(* Logix 5000 project; controller FPosB_EVO3_SP12 vendor 1 type 14 code 154 rev 30.11; software revision 30.01 *)
// v6: Studio5k 30+
// Works with CPX-E FW 1.1.24

TASK MainTask (continuous, watchdog 500 ms) : MainProgram

MODULES
   Local : vendor 1 type 14 code 154 (PointIO 0, rev 30.11)
      FMCP_Multi_EVO3_SP12 : ETHERNET-MODULE (Ethernet 192.168.4.20, rev 1.1, Output RPI 10 ms)
      Discrete_IO : Embedded (PointIO 1, rev 30.11, Output RPI 20 ms)
END_MODULES

ADD_ON_INSTRUCTION FMCP_Multi_EVO3_CPX_E_SP12_CPX_E   (* revision 3.14 15, vendor Festo Inc *)
// Multikinematic AOI to control up to 4 axis per kinematic and up to 3 different kinematics
// Revision note:
// 3.14.15: Multikinematic with 4 axis per kinematic
// 3.14.15: Additional tag to try to recover from a minor fault
VAR_IN_OUT
   InputData : DINT[64]; {required}
   OutputData : DINT[64]; {required}
END_VAR
VAR_INPUT
   K_I_N_E_M_A_T_I_C_1 : BOOL; {visible}
   I_n_p_u_t_s_K_1 : BOOL; {visible}
   sModeSelectorK1 : SINT; {visible}
END_VAR
VAR_OUTPUT
   sModeSelectedK1 : SINT; {visible}
END_VAR
VAR_INPUT
   rXAxisMove_CNCOffsetK1 : DINT; {visible}
   rYAxisMove_CNCOffsetK1 : DINT; {visible}
   rZAxisMove_CNCOffsetK1 : DINT; {visible}
   rUAxisMoveK1 : DINT; {visible}
   rZAxisOffset_CNCNumberK1 : DINT; {visible}
   rSmoothRad_CNCPhiK1 : DINT; {visible}
   rNominalVel_CNCConstantVelK1 : DINT := 1000; {visible}
   rLowVelMoveK1 : DINT := 100; {visible}
   rMoveAccelerationK1 : DINT := 1000; {visible}
   rMoveDecelerationK1 : DINT := 1000; {visible}
   rZAxisUpMoveK1 : DINT; {visible}
   bMoveK1 : BOOL; {visible}
   bJogXPosK1 : BOOL; {visible}
   bJogXNegK1 : BOOL; {visible}
   bJogYPosK1 : BOOL; {visible}
   bJogYNegK1 : BOOL; {visible}
   bJogZPosK1 : BOOL; {visible}
   bJogZNegK1 : BOOL; {visible}
   bJogUPosK1 : BOOL; {visible}
   bJogUNegK1 : BOOL; {visible}
   bAckMK1 : BOOL; {visible}
   bAckAllMK1 : BOOL; {visible}
   bHaltK1 : BOOL; {visible}
   bAbortMotionTaskK1 : BOOL; {visible}
   bTryToClearFaultK1 : BOOL; {visible}
   uOverrideK1 : DINT; {visible}
   O_u_t_p_u_t_s_K_1 : BOOL; {visible}
END_VAR
VAR_OUTPUT
   rXAxisActualPositionK1 : DINT; {visible}
   rYAxisActualPositionK1 : DINT; {visible}
   rZAxisActualPositionK1 : DINT; {visible}
   rUAxisActualPositionK1 : DINT; {visible}
   bEnabledK1 : BOOL; {visible}
   bHomedK1 : BOOL; {visible}
   bHaltedK1 : BOOL; {visible}
   bMoveDnK1 : BOOL; {visible}
   bMovingK1 : BOOL; {visible}
   bBusyK1 : BOOL; {visible}
   bErrorK1 : BOOL; {visible}
   bSafetyStatusK1 : BOOL; {visible}
   bMotionTaskAbortedK1 : BOOL; {visible}
   bXAxisSWLimitNegK1 : BOOL; {visible}
   bXAxisSWLimitPosK1 : BOOL; {visible}
   bYAxisSWLimitNegK1 : BOOL; {visible}
   bYAxisSWLimitPosK1 : BOOL; {visible}
   bZAxisSWLimitNegK1 : BOOL; {visible}
   bZAxisSWLimitPosK1 : BOOL; {visible}
   bUAxisSWLimitNegK1 : BOOL; {visible}
   bUAxisSWLimitPosK1 : BOOL; {visible}
   bHSwitchPoint1K1 : BOOL; {visible}
   bHSwitchPoint2K1 : BOOL; {visible}
   bMActiveK1 : BOOL; {visible}
   dErrorCode1K1 : DINT; {visible}
   dErrorCode2K1 : DINT; {visible}
   rGCodeLineK1 : DINT; {visible}
   bAtPrePickK1 : BOOL; {visible}
   bAtPickK1 : BOOL; {visible}
   bAtPrePlaceK1 : BOOL; {visible}
   bAtPlaceK1 : BOOL; {visible}
END_VAR
VAR_INPUT
   K_I_N_E_M_A_T_I_C_2 : BOOL; {visible}
   I_n_p_u_t_s_K_2 : BOOL; {visible}
   sModeSelectorK2 : SINT; {visible}
END_VAR
VAR_OUTPUT
   sModeSelectedK2 : SINT; {visible}
END_VAR
VAR_INPUT
   rXAxisMove_CNCOffsetK2 : DINT;
   rYAxisMove_CNCOffsetK2 : DINT; {visible}
   rZAxisMove_CNCOffsetK2 : DINT; {visible}
   rUAxisMoveK2 : DINT;
   rZAxisOffset_CNCNumberK2 : DINT; {visible}
   rSmoothRad_CNCPhiK2 : DINT; {visible}
   rNominalVel_CNCConstantVelK2 : DINT := 1000; {visible}
   rLowVelMoveK2 : DINT := 100; {visible}
   rMoveAccelerationK2 : DINT := 1000; {visible}
   rMoveDecelerationK2 : DINT := 1000; {visible}
   rZAxisUpMoveK2 : DINT; {visible}
   bMoveK2 : BOOL; {visible}
   bJogXPosK2 : BOOL; {visible}
   bJogXNegK2 : BOOL; {visible}
   bJogYPosK2 : BOOL; {visible}
   bJogYNegK2 : BOOL; {visible}
   bJogZPosK2 : BOOL; {visible}
   bJogZNegK2 : BOOL; {visible}
   bJogUPosK2 : BOOL; {visible}
   bJogUNegK2 : BOOL; {visible}
   bAckMK2 : BOOL; {visible}
   bAckAllMK2 : BOOL; {visible}
   bHaltK2 : BOOL; {visible}
   bAbortMotionTaskK2 : BOOL; {visible}
   bTryToClearFaultK2 : BOOL; {visible}
   uOverrideK2 : DINT; {visible}
   O_u_t_p_u_t_s_K_2 : BOOL; {visible}
END_VAR
VAR_OUTPUT
   rXAxisActualPositionK2 : DINT;
   rYAxisActualPositionK2 : DINT; {visible}
   rZAxisActualPositionK2 : DINT; {visible}
   rUAxisActualPositionK2 : DINT;
   bEnabledK2 : BOOL; {visible}
   bHomedK2 : BOOL; {visible}
   bHaltedK2 : BOOL; {visible}
   bMoveDnK2 : BOOL; {visible}
   bMovingK2 : BOOL; {visible}
   bBusyK2 : BOOL; {visible}
   bErrorK2 : BOOL; {visible}
   bSafetyStatusK2 : BOOL; {visible}
   bMotionTaskAbortedK2 : BOOL; {visible}
   bXAxisSWLimitNegK2 : BOOL; {visible}
   bXAxisSWLimitPosK2 : BOOL; {visible}
   bYAxisSWLimitNegK2 : BOOL; {visible}
   bYAxisSWLimitPosK2 : BOOL; {visible}
   bZAxisSWLimitNegK2 : BOOL; {visible}
   bZAxisSWLimitPosK2 : BOOL; {visible}
   bUAxisSWLimitNegK2 : BOOL; {visible}
   bUAxisSWLimitPosK2 : BOOL; {visible}
   bHSwitchPoint1K2 : BOOL; {visible}
   bHSwitchPoint2K2 : BOOL; {visible}
   bMActiveK2 : BOOL; {visible}
   dErrorCode1K2 : DINT; {visible}
   dErrorCode2K2 : DINT; {visible}
   rGCodeLineK2 : DINT; {visible}
   bAtPrePickK2 : BOOL; {visible}
   bAtPickK2 : BOOL; {visible}
   bAtPrePlaceK2 : BOOL; {visible}
   bAtPlaceK2 : BOOL; {visible}
END_VAR
VAR_INPUT
   K_I_N_E_M_A_T_I_C_3 : BOOL; {visible}
   I_n_p_u_t_s_K_3 : BOOL; {visible}
   sModeSelectorK3 : SINT; {visible}
END_VAR
VAR_OUTPUT
   sModeSelectedK3 : SINT; {visible}
END_VAR
VAR_INPUT
   rXAxisMove_CNCOffsetK3 : DINT; {visible}
   rYAxisMove_CNCOffsetK3 : DINT; {visible}
   rZAxisMove_CNCOffsetK3 : DINT; {visible}
   rUAxisMoveK3 : DINT; {visible}
   rZAxisOffset_CNCNumberK3 : DINT; {visible}
   rSmoothRad_CNCPhiK3 : DINT; {visible}
   rNominalVel_CNCConstantVelK3 : DINT := 1000; {visible}
   rLowVelMoveK3 : DINT := 100; {visible}
   rMoveAccelerationK3 : DINT := 1000; {visible}
   rMoveDecelerationK3 : DINT := 1000; {visible}
   rZAxisUpMoveK3 : DINT; {visible}
   bMoveK3 : BOOL; {visible}
   bJogXPosK3 : BOOL; {visible}
   bJogXNegK3 : BOOL; {visible}
   bJogYPosK3 : BOOL; {visible}
   bJogYNegK3 : BOOL; {visible}
   bJogZPosK3 : BOOL; {visible}
   bJogZNegK3 : BOOL; {visible}
   bJogUPosK3 : BOOL; {visible}
   bJogUNegK3 : BOOL; {visible}
   bAckMK3 : BOOL; {visible}
   bAckAllMK3 : BOOL; {visible}
   bHaltK3 : BOOL; {visible}
   bAbortMotionTaskK3 : BOOL; {visible}
   bTryToClearFaultK3 : BOOL; {visible}
   uOverrideK3 : DINT; {visible}
   O_u_t_p_u_t_s_K_3 : BOOL; {visible}
END_VAR
VAR_OUTPUT
   rXAxisActualPositionK3 : DINT; {visible}
   rYAxisActualPositionK3 : DINT; {visible}
   rZAxisActualPositionK3 : DINT; {visible}
   rUAxisActualPositionK3 : DINT; {visible}
   bEnabledK3 : BOOL; {visible}
   bHomedK3 : BOOL; {visible}
   bHaltedK3 : BOOL; {visible}
   bMoveDnK3 : BOOL; {visible}
   bMovingK3 : BOOL; {visible}
   bBusyK3 : BOOL; {visible}
   bErrorK3 : BOOL; {visible}
   bSafetyStatusK3 : BOOL; {visible}
   bMotionTaskAbortedK3 : BOOL; {visible}
   bXAxisSWLimitNegK3 : BOOL; {visible}
   bXAxisSWLimitPosK3 : BOOL; {visible}
   bYAxisSWLimitNegK3 : BOOL; {visible}
   bYAxisSWLimitPosK3 : BOOL; {visible}
   bZAxisSWLimitNegK3 : BOOL; {visible}
   bZAxisSWLimitPosK3 : BOOL; {visible}
   bUAxisSWLimitNegK3 : BOOL; {visible}
   bUAxisSWLimitPosK3 : BOOL; {visible}
   bHSwitchPoint1K3 : BOOL; {visible}
   bHSwitchPoint2K3 : BOOL; {visible}
   bMActiveK3 : BOOL; {visible}
   dErrorCode1K3 : DINT; {visible}
   dErrorCode2K3 : DINT; {visible}
   rGCodeLineK3 : DINT; {visible}
   bAtPrePickK3 : BOOL; {visible}
   bAtPickK3 : BOOL; {visible}
   bAtPrePlaceK3 : BOOL; {visible}
   bAtPlaceK3 : BOOL; {visible}
   O_t_h_e_r_s : BOOL; {visible}
   bFuseBlockStatus1 : BOOL; {visible}
   bFuseBlockStatus2 : BOOL; {visible}
   bFuseBlockStatus3 : BOOL; {visible}
END_VAR
VAR
   iErrorCodeLocal : DINT; {access None}
   EIP_Out_32 : DINT; {access None}
   EIP_Out_1 : DINT; {access None}
   EIP_In_0 : DINT; {access None}
   EIP_In_32 : DINT; {access None}
   EIP_Out_0 : DINT; {access None}
   EIP_Out_38 : DINT; {access None}
   EIP_Out_33 : DINT; {access None}
   EIP_Out_17 : DINT; {access None}
   EIP_Out_16 : DINT; {access None}
   EIP_Out_7 : DINT; {access None}
   EIP_Out_6 : DINT; {access None}
   EIP_In_16 : DINT; {access None}
   EIP_Out_39 : DINT; {access None}
   EIP_Out_23 : DINT; {access None}
   EIP_Out_22 : DINT; {access None}
END_VAR

ROUTINE Logic   (* structured text *)
   (*
   ***************************************************************************************************************************
   Name: FMCP Multikinematic Function Block
   Author: ca0lop
   Notes:
   Uses the X8 port to transfer mapped data to and from an AB PLC as fast as 10ms, 32I - 32O Data REAL.
   Festo Positioning Basic EVO3 V3.5.10.x Festo Position Basic Library with CoDeSys SP12
   *************2***************************************************************************************************************
   (*DataOut means Coming from PLC*)
   (*DataIn means Going to PLC*)
   (*FROM FESTO PLC X8*)
   EIP_In_0.0 := sModeSelectorK1.0;
   EIP_In_0.1 := sModeSelectorK1.1;
   EIP_In_0.2 := sModeSelectorK1.2;
   EIP_In_0.3 := sModeSelectorK1.3;
   EIP_In_0.4 := sModeSelectorK1.4;
   EIP_In_0.5 := sModeSelectorK1.5;
   EIP_In_0.6 := sModeSelectorK1.6;
   EIP_In_0.7 := sModeSelectorK1.7;
   EIP_In_0.8 := bHaltK1;
   EIP_In_0.9 := bAbortMotionTaskK1;
   EIP_In_0.10 := bMoveK1;
   EIP_In_0.11 := bJogXPosK1;
   EIP_In_0.12 := bJogXNegK1;
   EIP_In_0.13 := bJogYPosK1;
   EIP_In_0.14 := bJogYNegK1;
   EIP_In_0.15 := bJogZPosK1;
   EIP_In_0.16 := bJogZNegK1;
   EIP_In_0.17 := bJogUPosK1;
   EIP_In_0.18 := bJogUNegK1;
   EIP_In_0.19 := bAckMK1;
   EIP_In_0.20 := bAckAllMK1;
   EIP_In_0.21 := bTryToClearFaultK1;
   EIP_In_0.22 := 0;//SPARE
   EIP_In_0.23 := 0;//SPARE
   EIP_In_0.24 := uOverrideK1.0;
   EIP_In_0.25 := uOverrideK1.1;
   EIP_In_0.26 := uOverrideK1.2;
   EIP_In_0.27 := uOverrideK1.3;
   EIP_In_0.28 := uOverrideK1.4;
   EIP_In_0.29 := uOverrideK1.5;
   EIP_In_0.30 := uOverrideK1.6;
   EIP_In_0.31 := uOverrideK1.7;
   CPS(EIP_In_0,OutputData[0],1);
   
   OutputData[1] 	:= rXAxisMove_CNCOffsetK1;
   OutputData[2] 	:= rYAxisMove_CNCOffsetK1;
   OutputData[3] 	:= rZAxisMove_CNCOffsetK1;
   OutputData[4] 	:= rUAxisMoveK1;
   OutputData[5] 	:= rZAxisOffset_CNCNumberK1;
   OutputData[6] 	:= rSmoothRad_CNCPhiK1;
   OutputData[7] 	:= rNominalVel_CNCConstantVelK1;
   OutputData[8] 	:= rLowVelMoveK1;
   OutputData[9] 	:= rMoveAccelerationK1;
   OutputData[10]	:= rMoveDecelerationK1;
   OutputData[11] 	:= rZAxisUpMoveK1;
   OutputData[12] 	:= 0;//SPARE
   OutputData[13] 	:= 0;//SPARE
   OutputData[14] 	:= 0;//SPARE
   OutputData[15] 	:= 0;//SPARE
   
   
   EIP_In_16.0 := sModeSelectorK2.0;
   EIP_In_16.1 := sModeSelectorK2.1;
   EIP_In_16.2 := sModeSelectorK2.2;
   EIP_In_16.3 := sModeSelectorK2.3;
   EIP_In_16.4 := sModeSelectorK2.4;
   EIP_In_16.5 := sModeSelectorK2.5;
   EIP_In_16.6 := sModeSelectorK2.6;
   EIP_In_16.7 := sModeSelectorK2.7;
   EIP_In_16.8 := bHaltK2;
   EIP_In_16.9 := bAbortMotionTaskK2;
   EIP_In_16.10 := bMoveK2;
   EIP_In_16.11 := bJogXPosK2;
   EIP_In_16.12 := bJogXNegK2;
   EIP_In_16.13 := bJogYPosK2;
   EIP_In_16.14 := bJogYNegK2;
   EIP_In_16.15 := bJogZPosK2;
   EIP_In_16.16 := bJogZNegK2;
   EIP_In_16.17 := bJogUPosK2;
   EIP_In_16.18 := bJogUNegK2;
   EIP_In_16.19 := bAckMK2;
   EIP_In_16.20 := bAckAllMK2;
   EIP_In_16.21 := bTryToClearFaultK2;
   EIP_In_16.22 := 0;//SPARE
   EIP_In_16.23 := 0;//SPARE
   EIP_In_16.24 := uOverrideK2.0;
   EIP_In_16.25 := uOverrideK2.1;
   EIP_In_16.26 := uOverrideK2.2;
   EIP_In_16.27 := uOverrideK2.3;
   EIP_In_16.28 := uOverrideK2.4;
   EIP_In_16.29 := uOverrideK2.5;
   EIP_In_16.30 := uOverrideK2.6;
   EIP_In_16.31 := uOverrideK2.7;
   CPS(EIP_In_16,OutputData[16],1);
   
   OutputData[17] 	:= rXAxisMove_CNCOffsetK2;
   OutputData[18] 	:= rYAxisMove_CNCOffsetK2;
   OutputData[19] 	:= rZAxisMove_CNCOffsetK2;
   OutputData[20] 	:= rUAxisMoveK2;
   OutputData[21] 	:= rZAxisOffset_CNCNumberK2;
   OutputData[22] 	:= rSmoothRad_CNCPhiK2;
   OutputData[23] 	:= rNominalVel_CNCConstantVelK2;
   OutputData[24] 	:= rLowVelMoveK2;
   OutputData[25] 	:= rMoveAccelerationK2;
   OutputData[26]	:= rMoveDecelerationK2;
   OutputData[27] 	:= rZAxisUpMoveK2;
   OutputData[28] 	:= 0;//SPARE
   OutputData[29] 	:= 0;//SPARE
   OutputData[30] 	:= 0;//SPARE
   OutputData[31] 	:= 0;//SPARE
   
   EIP_In_32.0 := sModeSelectorK3.0;
   EIP_In_32.1 := sModeSelectorK3.1;
   EIP_In_32.2 := sModeSelectorK3.2;
   EIP_In_32.3 := sModeSelectorK3.3;
   EIP_In_32.4 := sModeSelectorK3.4;
   EIP_In_32.5 := sModeSelectorK3.5;
   EIP_In_32.6 := sModeSelectorK3.6;
   EIP_In_32.7 := sModeSelectorK3.7;
   EIP_In_32.8 := bHaltK3;
   EIP_In_32.9 := bAbortMotionTaskK3;
   EIP_In_32.10 := bMoveK3;
   EIP_In_32.11 := bJogXPosK3;
   EIP_In_32.12 := bJogXNegK3;
   EIP_In_32.13 := bJogYPosK3;
   EIP_In_32.14 := bJogYNegK3;
   EIP_In_32.15 := bJogZPosK3;
   EIP_In_32.16 := bJogZNegK3;
   EIP_In_32.17 := bJogUPosK3;
   EIP_In_32.18 := bJogUNegK3;
   EIP_In_32.19 := bAckMK3;
   EIP_In_32.20 := bAckAllMK3;
   EIP_In_32.21 := bTryToClearFaultK3;
   EIP_In_32.22 := 0;//SPARE
   EIP_In_32.23 := 0;//SPARE
   EIP_In_32.24 := uOverrideK3.0;
   EIP_In_32.25 := uOverrideK3.1;
   EIP_In_32.26 := uOverrideK3.2;
   EIP_In_32.27 := uOverrideK3.3;
   EIP_In_32.28 := uOverrideK3.4;
   EIP_In_32.29 := uOverrideK3.5;
   EIP_In_32.30 := uOverrideK3.6;
   EIP_In_32.31 := uOverrideK3.7;
   CPS(EIP_In_32,OutputData[32],1);
   
   OutputData[33] 	:= rXAxisMove_CNCOffsetK3;
   OutputData[34] 	:= rYAxisMove_CNCOffsetK3;
   OutputData[35] 	:= rZAxisMove_CNCOffsetK3;
   OutputData[36] 	:= rUAxisMoveK3;
   OutputData[37] 	:= rZAxisOffset_CNCNumberK3;
   OutputData[38] 	:= rSmoothRad_CNCPhiK3;
   OutputData[39] 	:= rNominalVel_CNCConstantVelK3;
   OutputData[40] 	:= rLowVelMoveK3;
   OutputData[41] 	:= rMoveAccelerationK3;
   OutputData[42]	:= rMoveDecelerationK3;
   OutputData[43] 	:= rZAxisUpMoveK3;
   OutputData[44] 	:= 0;//SPARE
   OutputData[45] 	:= 0;//SPARE
   OutputData[46] 	:= 0;//SPARE
   OutputData[47] 	:= 0;//SPARE
   OutputData[48] 	:= 0;//SPARE
   OutputData[49] 	:= 0;//SPARE
   OutputData[50] 	:= 0;//SPARE
   OutputData[51] 	:= 0;//SPARE
   OutputData[52] 	:= 0;//SPARE
   OutputData[53] 	:= 0;//SPARE
   OutputData[54] 	:= 0;//SPARE
   OutputData[55] 	:= 0;//SPARE
   OutputData[56] 	:= 0;//SPARE
   OutputData[57] 	:= 0;//SPARE
   OutputData[58] 	:= 0;//SPARE
   OutputData[59] 	:= 0;//SPARE
   OutputData[60] 	:= 0;//SPARE
   OutputData[61] 	:= 0;//SPARE
   OutputData[62] 	:= 0;//SPARE
   OutputData[63] 	:= 0;//SPARE
   
   
   (*===============================================================================================================================================*)
   (*===============================================================================================================================================*)
   (*===============================================================================================================================================*)
   (*===============================================================================================================================================*)
   (*===============================================================================================================================================*)
   (*===============================================================================================================================================*)
   (*===============================================================================================================================================*)
   
   (*TO FESTO PLC X8*)
   CPS(InputData[0],EIP_Out_0,1);
   sModeSelectedK1.0 		:= EIP_Out_0.0;
   sModeSelectedK1.1 		:= EIP_Out_0.1;
   sModeSelectedK1.2 		:= EIP_Out_0.2;
   sModeSelectedK1.3 		:= EIP_Out_0.3;
   sModeSelectedK1.4 		:= EIP_Out_0.4;
   sModeSelectedK1.5 		:= EIP_Out_0.5;
   sModeSelectedK1.6 		:= EIP_Out_0.6;
   sModeSelectedK1.7 		:= EIP_Out_0.7;
   bSafetyStatusK1 		:= EIP_Out_0.8;
   bMotionTaskAbortedK1 	:= EIP_Out_0.9;
   bEnabledK1 				:= EIP_Out_0.10;
   bHomedK1 				:= EIP_Out_0.11;
   bHaltedK1 				:= EIP_Out_0.12;
   bMoveDnK1 				:= EIP_Out_0.13;
   bMovingK1 				:= EIP_Out_0.14;
   bBusyK1 				:= EIP_Out_0.15;
   bErrorK1 				:= EIP_Out_0.16;
   bXAxisSWLimitNegK1 		:= EIP_Out_0.17;
   bXAxisSWLimitPosK1 		:= EIP_Out_0.18;
   bYAxisSWLimitNegK1 		:= EIP_Out_0.19;
   bYAxisSWLimitPosK1 		:= EIP_Out_0.20;
   bZAxisSWLimitNegK1 		:= EIP_Out_0.21;
   bZAxisSWLimitPosK1 		:= EIP_Out_0.22;
   bUAxisSWLimitNegK1 		:= EIP_Out_0.23;
   bUAxisSWLimitPosK1 		:= EIP_Out_0.24;
   bHSwitchPoint1K1 		:= EIP_Out_0.25;
   bHSwitchPoint2K1 		:= EIP_Out_0.26;
   bMActiveK1 				:= EIP_Out_0.27;
   bAtPrePickK1 			:= EIP_Out_0.28;
   bAtPickK1 				:= EIP_Out_0.29;
   bAtPrePlaceK1 			:= EIP_Out_0.30;
   bAtPlaceK1 				:= EIP_Out_0.31;
   //CPS(InputData[1],EIP_Out_1,1); //SPARE
   rXAxisActualPositionK1	:= InputData[2];
   rYAxisActualPositionK1	:= InputData[3];
   rZAxisActualPositionK1	:= InputData[4];
   rUAxisActualPositionK1	:= InputData[5];
   
   (*Last two errors listed below*)
   CPS(InputData[6],EIP_Out_6,1);
   dErrorCode1K1.0 := EIP_Out_6.0;
   dErrorCode1K1.1 := EIP_Out_6.1;
   dErrorCode1K1.2 := EIP_Out_6.2;
   dErrorCode1K1.3 := EIP_Out_6.3;
   dErrorCode1K1.4 := EIP_Out_6.4;
   dErrorCode1K1.5 := EIP_Out_6.5;
   dErrorCode1K1.6 := EIP_Out_6.6;
   dErrorCode1K1.7 := EIP_Out_6.7;
   dErrorCode1K1.8 := EIP_Out_1.8;
   dErrorCode1K1.9 := EIP_Out_6.9;
   dErrorCode1K1.10 := EIP_Out_6.10;
   dErrorCode1K1.11 := EIP_Out_6.11;
   dErrorCode1K1.12 := EIP_Out_6.12;
   dErrorCode1K1.13 := EIP_Out_6.13;
   dErrorCode1K1.14 := EIP_Out_6.14;
   dErrorCode1K1.15 := EIP_Out_6.15;
   dErrorCode1K1.16 := EIP_Out_6.16;
   dErrorCode1K1.17 := EIP_Out_6.17;
   dErrorCode1K1.18 := EIP_Out_6.18;
   dErrorCode1K1.19 := EIP_Out_6.19;
   dErrorCode1K1.20 := EIP_Out_6.20;
   dErrorCode1K1.21 := EIP_Out_6.21;
   dErrorCode1K1.22 := EIP_Out_6.22;
   dErrorCode1K1.23 := EIP_Out_6.23;
   dErrorCode1K1.24 := EIP_Out_6.24;
   dErrorCode1K1.25 := EIP_Out_6.25;
   dErrorCode1K1.26 := EIP_Out_6.26;
   dErrorCode1K1.27 := EIP_Out_6.27;
   dErrorCode1K1.28 := EIP_Out_6.28;
   dErrorCode1K1.29 := EIP_Out_6.29;
   dErrorCode1K1.30 := EIP_Out_6.30;
   dErrorCode1K1.31 := EIP_Out_6.31;
   
   CPS(InputData[7],EIP_Out_7,1);
   dErrorCode2K1.0 := EIP_Out_7.0;
   dErrorCode2K1.1 := EIP_Out_7.1;
   dErrorCode2K1.2 := EIP_Out_7.2;
   dErrorCode2K1.3 := EIP_Out_7.3;
   dErrorCode2K1.4 := EIP_Out_7.4;
   dErrorCode2K1.5 := EIP_Out_7.5;
   dErrorCode2K1.6 := EIP_Out_7.6;
   dErrorCode2K1.7 := EIP_Out_7.7;
   dErrorCode2K1.8 := EIP_Out_7.8;
   dErrorCode2K1.9 := EIP_Out_7.9;
   dErrorCode2K1.10 := EIP_Out_7.10;
   dErrorCode2K1.11 := EIP_Out_7.11;
   dErrorCode2K1.12 := EIP_Out_7.12;
   dErrorCode2K1.13 := EIP_Out_7.13;
   dErrorCode2K1.14 := EIP_Out_7.14;
   dErrorCode2K1.15 := EIP_Out_7.15;
   dErrorCode2K1.16 := EIP_Out_7.16;
   dErrorCode2K1.17 := EIP_Out_7.17;
   dErrorCode2K1.18 := EIP_Out_7.18;
   dErrorCode2K1.19 := EIP_Out_7.19;
   dErrorCode2K1.20 := EIP_Out_7.20;
   dErrorCode2K1.21 := EIP_Out_7.21;
   dErrorCode2K1.22 := EIP_Out_7.22;
   dErrorCode2K1.23 := EIP_Out_7.23;
   dErrorCode2K1.24 := EIP_Out_7.24;
   dErrorCode2K1.25 := EIP_Out_7.25;
   dErrorCode2K1.26 := EIP_Out_7.26;
   dErrorCode2K1.27 := EIP_Out_7.27;
   dErrorCode2K1.28 := EIP_Out_7.28;
   dErrorCode2K1.29 := EIP_Out_7.29;
   dErrorCode2K1.30 := EIP_Out_7.30;
   dErrorCode2K1.31 := EIP_Out_7.31;
   
   rGCodeLineK1 := InputData[8];
   
   //CPS(InputData[9],EIP_Out_9,1); //SPARE
   //CPS(InputData[10],EIP_Out_10,1); //SPARE
   //CPS(InputData[11],EIP_Out_11,1); //SPARE
   //CPS(InputData[12],EIP_Out_12,1); //SPARE
   //CPS(InputData[13],EIP_Out_13,1); //SPARE
   //CPS(InputData[14],EIP_Out_14,1); //SPARE
   //CPS(InputData[15],EIP_Out_15,1); //SPARE
   
   CPS(InputData[16],EIP_Out_16,1);
   sModeSelectedK2.0 		:= EIP_Out_16.0;
   sModeSelectedK2.1 		:= EIP_Out_16.1;
   sModeSelectedK2.2 		:= EIP_Out_16.2;
   sModeSelectedK2.3 		:= EIP_Out_16.3;
   sModeSelectedK2.4 		:= EIP_Out_16.4;
   sModeSelectedK2.5 		:= EIP_Out_16.5;
   sModeSelectedK2.6 		:= EIP_Out_16.6;
   sModeSelectedK2.7 		:= EIP_Out_16.7;
   bSafetyStatusK2 		:= EIP_Out_16.8;
   bMotionTaskAbortedK2 	:= EIP_Out_16.9;
   bEnabledK2 				:= EIP_Out_16.10;
   bHomedK2 				:= EIP_Out_16.11;
   bHaltedK2 				:= EIP_Out_16.12;
   bMoveDnK2 				:= EIP_Out_16.13;
   bMovingK2 				:= EIP_Out_16.14;
   bBusyK2 				:= EIP_Out_16.15;
   bErrorK2 				:= EIP_Out_16.16;
   bXAxisSWLimitNegK2 		:= EIP_Out_16.17;
   bXAxisSWLimitPosK2 		:= EIP_Out_16.18;
   bYAxisSWLimitNegK2 		:= EIP_Out_16.19;
   bYAxisSWLimitPosK2 		:= EIP_Out_16.20;
   bZAxisSWLimitNegK2 		:= EIP_Out_16.21;
   bZAxisSWLimitPosK2 		:= EIP_Out_16.22;
   bUAxisSWLimitNegK2 		:= EIP_Out_16.23;
   bUAxisSWLimitPosK2 		:= EIP_Out_16.24;
   bHSwitchPoint1K2 		:= EIP_Out_16.25;
   bHSwitchPoint2K2 		:= EIP_Out_16.26;
   bMActiveK2 				:= EIP_Out_16.27;
   bAtPrePickK2 			:= EIP_Out_16.28;
   bAtPickK2 				:= EIP_Out_16.29;
   bAtPrePlaceK2 			:= EIP_Out_16.30;
   bAtPlaceK2 				:= EIP_Out_16.31;
   
   //CPS(InputData[17],EIP_Out_17,1); //SPARE
   
   rXAxisActualPositionK2	:= InputData[18];
   rYAxisActualPositionK2	:= InputData[19];
   rZAxisActualPositionK2	:= InputData[20];
   rUAxisActualPositionK2	:= InputData[21];
   
   (*Last two errors listed below*)
   CPS(InputData[22],EIP_Out_22,1);
   dErrorCode1K2.0 := EIP_Out_22.0;
   dErrorCode1K2.1 := EIP_Out_22.1;
   dErrorCode1K2.2 := EIP_Out_22.2;
   dErrorCode1K2.3 := EIP_Out_22.3;
   dErrorCode1K2.4 := EIP_Out_22.4;
   dErrorCode1K2.5 := EIP_Out_22.5;
   dErrorCode1K2.6 := EIP_Out_22.6;
   dErrorCode1K2.7 := EIP_Out_22.7;
   dErrorCode1K2.8 := EIP_Out_1.8;
   dErrorCode1K2.9 := EIP_Out_22.9;
   dErrorCode1K2.10 := EIP_Out_22.10;
   dErrorCode1K2.11 := EIP_Out_22.11;
   dErrorCode1K2.12 := EIP_Out_22.12;
   dErrorCode1K2.13 := EIP_Out_22.13;
   dErrorCode1K2.14 := EIP_Out_22.14;
   dErrorCode1K2.15 := EIP_Out_22.15;
   dErrorCode1K2.16 := EIP_Out_22.16;
   dErrorCode1K2.17 := EIP_Out_22.17;
   dErrorCode1K2.18 := EIP_Out_22.18;
   dErrorCode1K2.19 := EIP_Out_22.19;
   dErrorCode1K2.20 := EIP_Out_22.20;
   dErrorCode1K2.21 := EIP_Out_22.21;
   dErrorCode1K2.22 := EIP_Out_22.22;
   dErrorCode1K2.23 := EIP_Out_22.23;
   dErrorCode1K2.24 := EIP_Out_22.24;
   dErrorCode1K2.25 := EIP_Out_22.25;
   dErrorCode1K2.26 := EIP_Out_22.26;
   dErrorCode1K2.27 := EIP_Out_22.27;
   dErrorCode1K2.28 := EIP_Out_22.28;
   dErrorCode1K2.29 := EIP_Out_22.29;
   dErrorCode1K2.30 := EIP_Out_22.30;
   dErrorCode1K2.31 := EIP_Out_22.31;
   
   CPS(InputData[23],EIP_Out_23,1);
   dErrorCode2K2.0 := EIP_Out_23.0;
   dErrorCode2K2.1 := EIP_Out_23.1;
   dErrorCode2K2.2 := EIP_Out_23.2;
   dErrorCode2K2.3 := EIP_Out_23.3;
   dErrorCode2K2.4 := EIP_Out_23.4;
   dErrorCode2K2.5 := EIP_Out_23.5;
   dErrorCode2K2.6 := EIP_Out_23.6;
   dErrorCode2K2.7 := EIP_Out_23.7;
   dErrorCode2K2.8 := EIP_Out_23.8;
   dErrorCode2K2.9 := EIP_Out_23.9;
   dErrorCode2K2.10 := EIP_Out_23.10;
   dErrorCode2K2.11 := EIP_Out_23.11;
   dErrorCode2K2.12 := EIP_Out_23.12;
   dErrorCode2K2.13 := EIP_Out_23.13;
   dErrorCode2K2.14 := EIP_Out_23.14;
   dErrorCode2K2.15 := EIP_Out_23.15;
   dErrorCode2K2.16 := EIP_Out_23.16;
   dErrorCode2K2.17 := EIP_Out_23.17;
   dErrorCode2K2.18 := EIP_Out_23.18;
   dErrorCode2K2.19 := EIP_Out_23.19;
   dErrorCode2K2.20 := EIP_Out_23.20;
   dErrorCode2K2.21 := EIP_Out_23.21;
   dErrorCode2K2.22 := EIP_Out_23.22;
   dErrorCode2K2.23 := EIP_Out_23.23;
   dErrorCode2K2.24 := EIP_Out_23.24;
   dErrorCode2K2.25 := EIP_Out_23.25;
   dErrorCode2K2.26 := EIP_Out_23.26;
   dErrorCode2K2.27 := EIP_Out_23.27;
   dErrorCode2K2.28 := EIP_Out_23.28;
   dErrorCode2K2.29 := EIP_Out_23.29;
   dErrorCode2K2.30 := EIP_Out_23.30;
   dErrorCode2K2.31 := EIP_Out_23.31;
   
   rGCodeLineK2 := InputData[24];
   
   //CPS(InputData[25],EIP_Out_25,1); //SPARE
   //CPS(InputData[26],EIP_Out_26,1); //SPARE
   //CPS(InputData[27],EIP_Out_27,1); //SPARE
   //CPS(InputData[28],EIP_Out_28,1); //SPARE
   //CPS(InputData[29],EIP_Out_29,1); //SPARE
   //CPS(InputData[30],EIP_Out_30,1); //SPARE
   //CPS(InputData[31],EIP_Out_31,1); //SPARE
   
   CPS(InputData[32],EIP_Out_32,1);
   sModeSelectedK3.0 		:= EIP_Out_32.0;
   sModeSelectedK3.1 		:= EIP_Out_32.1;
   sModeSelectedK3.2 		:= EIP_Out_32.2;
   sModeSelectedK3.3 		:= EIP_Out_32.3;
   sModeSelectedK3.4 		:= EIP_Out_32.4;
   sModeSelectedK3.5 		:= EIP_Out_32.5;
   sModeSelectedK3.6 		:= EIP_Out_32.6;
   sModeSelectedK3.7 		:= EIP_Out_32.7;
   bSafetyStatusK3 		:= EIP_Out_32.8;
   bMotionTaskAbortedK3 	:= EIP_Out_32.9;
   bEnabledK3 				:= EIP_Out_32.10;
   bHomedK3 				:= EIP_Out_32.11;
   bHaltedK3 				:= EIP_Out_32.12;
   bMoveDnK3 				:= EIP_Out_32.13;
   bMovingK3 				:= EIP_Out_32.14;
   bBusyK3 				:= EIP_Out_32.15;
   bErrorK3 				:= EIP_Out_32.16;
   bXAxisSWLimitNegK3 		:= EIP_Out_32.17;
   bXAxisSWLimitPosK3 		:= EIP_Out_32.18;
   bYAxisSWLimitNegK3 		:= EIP_Out_32.19;
   bYAxisSWLimitPosK3 		:= EIP_Out_32.20;
   bZAxisSWLimitNegK3 		:= EIP_Out_32.21;
   bZAxisSWLimitPosK3 		:= EIP_Out_32.22;
   bUAxisSWLimitNegK3 		:= EIP_Out_32.23;
   bUAxisSWLimitPosK3 		:= EIP_Out_32.24;
   bHSwitchPoint1K3 		:= EIP_Out_32.25;
   bHSwitchPoint2K3 		:= EIP_Out_32.26;
   bMActiveK3 				:= EIP_Out_32.27;
   bAtPrePickK3 			:= EIP_Out_32.28;
   bAtPickK3 				:= EIP_Out_32.29;
   bAtPrePlaceK3 			:= EIP_Out_32.30;
   bAtPlaceK3 				:= EIP_Out_32.31;
   
   //CPS(InputData[33],EIP_Out_33,1); //SPARE
   
   rXAxisActualPositionK3	:= InputData[34];
   rYAxisActualPositionK3	:= InputData[35];
   rZAxisActualPositionK3	:= InputData[36];
   rUAxisActualPositionK3	:= InputData[37];
   
   (*Last two errors listed below*)
   CPS(InputData[38],EIP_Out_38,1);
   dErrorCode1K3.0 := EIP_Out_38.0;
   dErrorCode1K3.1 := EIP_Out_38.1;
   dErrorCode1K3.2 := EIP_Out_38.2;
   dErrorCode1K3.3 := EIP_Out_38.3;
   dErrorCode1K3.4 := EIP_Out_38.4;
   dErrorCode1K3.5 := EIP_Out_38.5;
   dErrorCode1K3.6 := EIP_Out_38.6;
   dErrorCode1K3.7 := EIP_Out_38.7;
   dErrorCode1K3.8 := EIP_Out_1.8;
   dErrorCode1K3.9 := EIP_Out_38.9;
   dErrorCode1K3.10 := EIP_Out_38.10;
   dErrorCode1K3.11 := EIP_Out_38.11;
   dErrorCode1K3.12 := EIP_Out_38.12;
   dErrorCode1K3.13 := EIP_Out_38.13;
   dErrorCode1K3.14 := EIP_Out_38.14;
   dErrorCode1K3.15 := EIP_Out_38.15;
   dErrorCode1K3.16 := EIP_Out_38.16;
   dErrorCode1K3.17 := EIP_Out_38.17;
   dErrorCode1K3.18 := EIP_Out_38.18;
   dErrorCode1K3.19 := EIP_Out_38.19;
   dErrorCode1K3.20 := EIP_Out_38.20;
   dErrorCode1K3.21 := EIP_Out_38.21;
   dErrorCode1K3.22 := EIP_Out_38.22;
   dErrorCode1K3.23 := EIP_Out_38.23;
   dErrorCode1K3.24 := EIP_Out_38.24;
   dErrorCode1K3.25 := EIP_Out_38.25;
   dErrorCode1K3.26 := EIP_Out_38.26;
   dErrorCode1K3.27 := EIP_Out_38.27;
   dErrorCode1K3.28 := EIP_Out_38.28;
   dErrorCode1K3.29 := EIP_Out_38.29;
   dErrorCode1K3.30 := EIP_Out_38.30;
   dErrorCode1K3.31 := EIP_Out_38.31;
   
   CPS(InputData[39],EIP_Out_39,1);
   dErrorCode2K3.0 := EIP_Out_39.0;
   dErrorCode2K3.1 := EIP_Out_39.1;
   dErrorCode2K3.2 := EIP_Out_39.2;
   dErrorCode2K3.3 := EIP_Out_39.3;
   dErrorCode2K3.4 := EIP_Out_39.4;
   dErrorCode2K3.5 := EIP_Out_39.5;
   dErrorCode2K3.6 := EIP_Out_39.6;
   dErrorCode2K3.7 := EIP_Out_39.7;
   dErrorCode2K3.8 := EIP_Out_39.8;
   dErrorCode2K3.9 := EIP_Out_39.9;
   dErrorCode2K3.10 := EIP_Out_39.10;
   dErrorCode2K3.11 := EIP_Out_39.11;
   dErrorCode2K3.12 := EIP_Out_39.12;
   dErrorCode2K3.13 := EIP_Out_39.13;
   dErrorCode2K3.14 := EIP_Out_39.14;
   dErrorCode2K3.15 := EIP_Out_39.15;
   dErrorCode2K3.16 := EIP_Out_39.16;
   dErrorCode2K3.17 := EIP_Out_39.17;
   dErrorCode2K3.18 := EIP_Out_39.18;
   dErrorCode2K3.19 := EIP_Out_39.19;
   dErrorCode2K3.20 := EIP_Out_39.20;
   dErrorCode2K3.21 := EIP_Out_39.21;
   dErrorCode2K3.22 := EIP_Out_39.22;
   dErrorCode2K3.23 := EIP_Out_39.23;
   dErrorCode2K3.24 := EIP_Out_39.24;
   dErrorCode2K3.25 := EIP_Out_39.25;
   dErrorCode2K3.26 := EIP_Out_39.26;
   dErrorCode2K3.27 := EIP_Out_39.27;
   dErrorCode2K3.28 := EIP_Out_39.28;
   dErrorCode2K3.29 := EIP_Out_39.29;
   dErrorCode2K3.30 := EIP_Out_39.30;
   dErrorCode2K3.31 := EIP_Out_39.31;
   
   rGCodeLineK3 := InputData[40];
   
   //CPS(InputData[41],EIP_Out_41,1); //SPARE
   //CPS(InputData[42],EIP_Out_42,1); //SPARE
   //CPS(InputData[43],EIP_Out_43,1); //SPARE
   //CPS(InputData[44],EIP_Out_44,1); //SPARE
   //CPS(InputData[45],EIP_Out_45,1); //SPARE
   //CPS(InputData[46],EIP_Out_46,1); //SPARE
   //CPS(InputData[47],EIP_Out_47,1); //SPARE
   
   //CPS(InputData[48],EIP_Out_48,1); //SPARE
   //CPS(InputData[49],EIP_Out_49,1); //SPARE
   //CPS(InputData[50],EIP_Out_50,1); //SPARE
   //CPS(InputData[51],EIP_Out_51,1); //SPARE
   //CPS(InputData[52],EIP_Out_52,1); //SPARE
   //CPS(InputData[53],EIP_Out_53,1); //SPARE
   //CPS(InputData[54],EIP_Out_54,1); //SPARE
   //CPS(InputData[55],EIP_Out_55,1); //SPARE
   //CPS(InputData[56],EIP_Out_56,1); //SPARE
   //CPS(InputData[57],EIP_Out_57,1); //SPARE
   //CPS(InputData[58],EIP_Out_58,1); //SPARE
   //CPS(InputData[59],EIP_Out_59,1); //SPARE
   //CPS(InputData[60],EIP_Out_60,1); //SPARE
   //CPS(InputData[61],EIP_Out_61,1); //SPARE
   //CPS(InputData[62],EIP_Out_62,1); //SPARE
   //CPS(InputData[63],EIP_Out_63,1); //SPARE
   
   
   
   
END_ROUTINE
END_ADD_ON_INSTRUCTION

VAR_GLOBAL   (* controller tags *)
   AAxisAdjustment : REAL;
   AccelDecel : REAL := 500.0;
   AlwaysON : BOOL;
   bAckMMode6wZOffset : BOOL;
   bContinue : BOOL;
   bDummy : BOOL;
   bMCR : BOOL;
   bMoveToCNC : BOOL;
   bMoveToHome : BOOL;
   bPauseBetweenPoints : BOOL;
   bStartMode5 : BOOL;
   bStartMode6woZOffset : BOOL;
   bStartMode6wZOffset : BOOL;
   bStartMode7 : BOOL;
   CNCConstantVelocity : DINT;
   CNCNumberToRun : REAL := 3.0;
   CNCOverride : DINT;
   CNCRotate : REAL;
   dDemoModeSelector : DINT := 9;
   FMCP_M : FMCP_Multi_EVO3_CPX_E_SP12_CPX_E := (bHomedK1 := 1, rGCodeLineK1 := -1, rGCodeLineK2 := -1, rNominalVel_CNCConstantVelK3 := 1000, rLowVelMoveK3 := 100, rMoveAccelerationK3 := 1000, rMoveDecelerationK3 := 1000);
   NominalVelocity : REAL := 3000.0;
   NominalVelocityCNC : DINT;
   OS0 : BOOL;
   OS1 : BOOL;
   OS10 : BOOL;
   OS11 : BOOL;
   rUAxisDemoTargetDestination : REAL := 200.0;
   rXAxisDemo_CNCOffset : REAL;
   rXAxisDemoTargetDestination : REAL := 10000.0;
   rYAxisDemo_CNCOffset : REAL;
   rYAxisDemoTargetDestination : REAL := 5000.0;
   rZAxisDemo_CNCOffset : REAL;
   rZAxisDemoTargetDestination : REAL := 1000.0;
   rZAxisOffsetDemoTargetDestination : REAL := 30.0;
   TONAbort : TIMER := (PRE := 500);
   XAxisAdjustment : REAL;
   YAxisAdjustment : REAL;
   ZAxisAdjustment : REAL;
END_VAR

PROGRAM MainProgram   (* main routine MainRoutine *)
VAR
   StepSeqMode5 : BOOL[32];
   StepSeqMode6wOffset : BOOL[32];
   StepSeqMode6woOffset : BOOL[32];
   StepSeqMode7CNC : BOOL[32];
END_VAR

ROUTINE MainRoutine   (* ladder *)
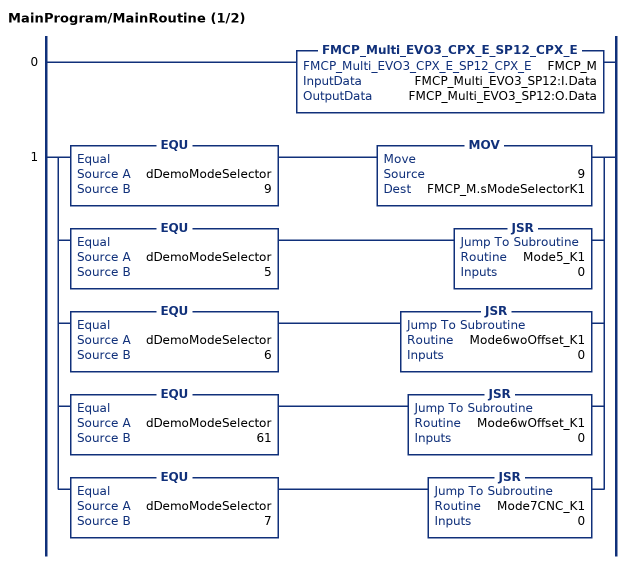
   0: FMCP_Multi_EVO3_CPX_E_SP12_CPX_E(FMCP_M,FMCP_Multi_EVO3_SP12:I.Data,FMCP_Multi_EVO3_SP12:O.Data);
   1: [EQU(dDemoModeSelector,9) MOV(9,FMCP_M.sModeSelectorK1) ,EQU(dDemoModeSelector,5) JSR(Mode5_K1,0) ,EQU(dDemoModeSelector,6) JSR(Mode6woOffset_K1,0) ,EQU(dDemoModeSelector,61) JSR(Mode6wOffset_K1,0) ,EQU(dDemoModeSelector,7) JSR(Mode7CNC_K1,0) ];
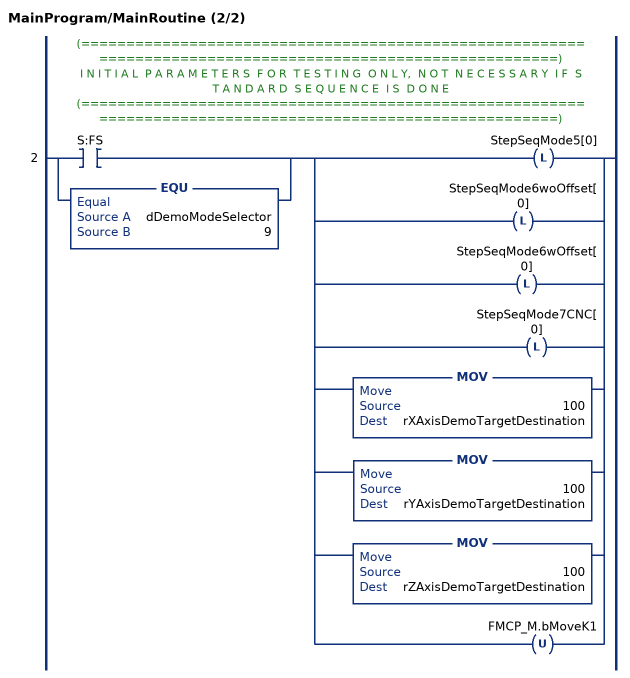
   // (===========================================================================================================)
   // I N I T I A L  P A R A M E T E R S  F O R  T E S T I N G  O N L Y,  N O T  N E C E S S A R Y  I F  S T A N D A R D  S E Q U E N C E  I S  D O N E
   // (===========================================================================================================)
   2: [XIC(S:FS) ,EQU(dDemoModeSelector,9) ][OTL(StepSeqMode5[0]) ,OTL(StepSeqMode6woOffset[0]) ,OTL(StepSeqMode6wOffset[0]) ,OTL(StepSeqMode7CNC[0]) ,MOV(100,rXAxisDemoTargetDestination) ,MOV(100,rYAxisDemoTargetDestination) ,MOV(100,rZAxisDemoTargetDestination) ,OTU(FMCP_M.bMoveK1) ];
END_ROUTINE

ROUTINE Mode5_K1   (* ladder *)
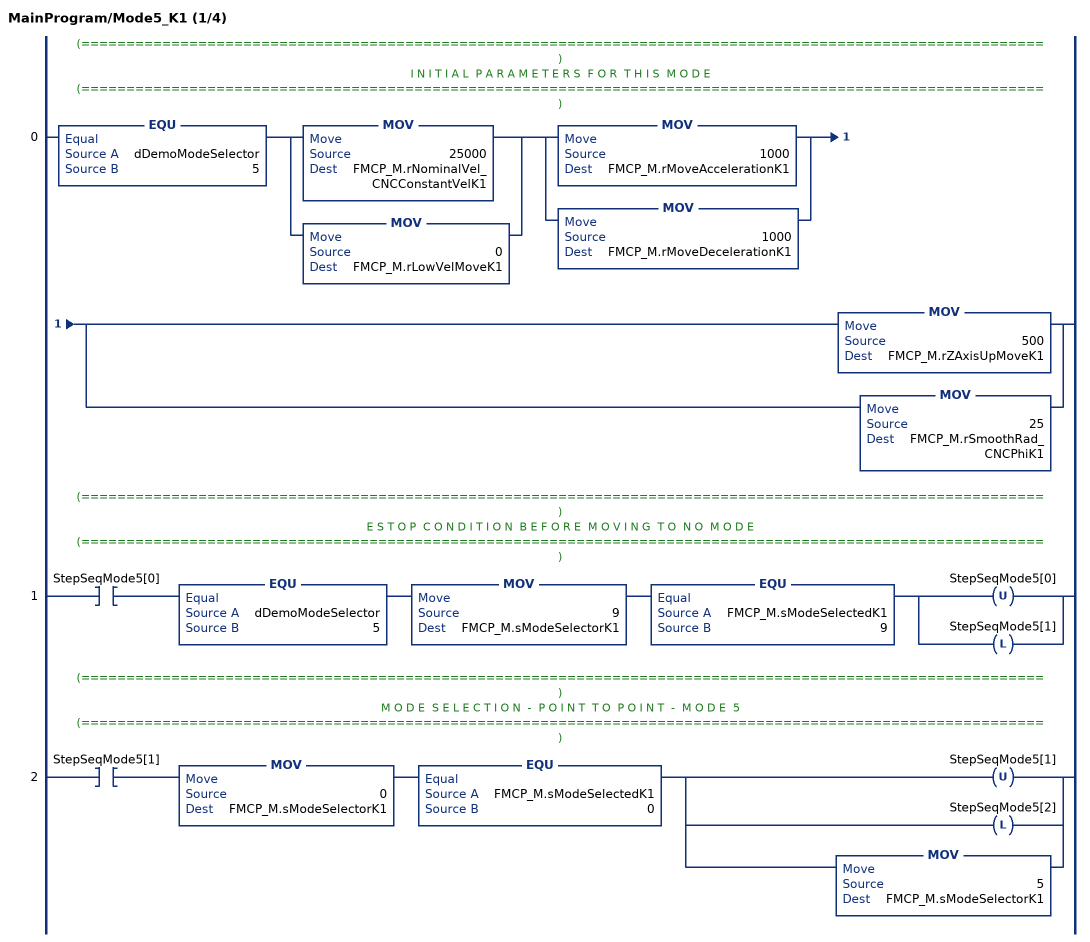
   // (===========================================================================================================)
   // I N I T I A L  P A R A M E T E R S  F O R  T H I S  M O D E
   // (===========================================================================================================)
   0: EQU(dDemoModeSelector,5)[MOV(25000,FMCP_M.rNominalVel_CNCConstantVelK1) ,MOV(0,FMCP_M.rLowVelMoveK1) ][MOV(1000,FMCP_M.rMoveAccelerationK1) ,MOV(1000,FMCP_M.rMoveDecelerationK1) ][MOV(500,FMCP_M.rZAxisUpMoveK1) ,MOV(25,FMCP_M.rSmoothRad_CNCPhiK1) ];
   // (===========================================================================================================)
   // E S T O P  C O N D I T I O N  B E F O R E  M O V I N G  T O  N O  M O D E
   // (===========================================================================================================)
   1: XIC(StepSeqMode5[0])EQU(dDemoModeSelector,5)MOV(9,FMCP_M.sModeSelectorK1)EQU(FMCP_M.sModeSelectedK1,9)[OTU(StepSeqMode5[0]) ,OTL(StepSeqMode5[1]) ];
   // (===========================================================================================================)
   // M O D E  S E L E C T I O N  -  P O I N T  T O  P O I N T  -  M O D E  5
   // (===========================================================================================================)
   2: XIC(StepSeqMode5[1])MOV(0,FMCP_M.sModeSelectorK1)EQU(FMCP_M.sModeSelectedK1,0)[OTU(StepSeqMode5[1]) ,OTL(StepSeqMode5[2]) ,MOV(5,FMCP_M.sModeSelectorK1) ];
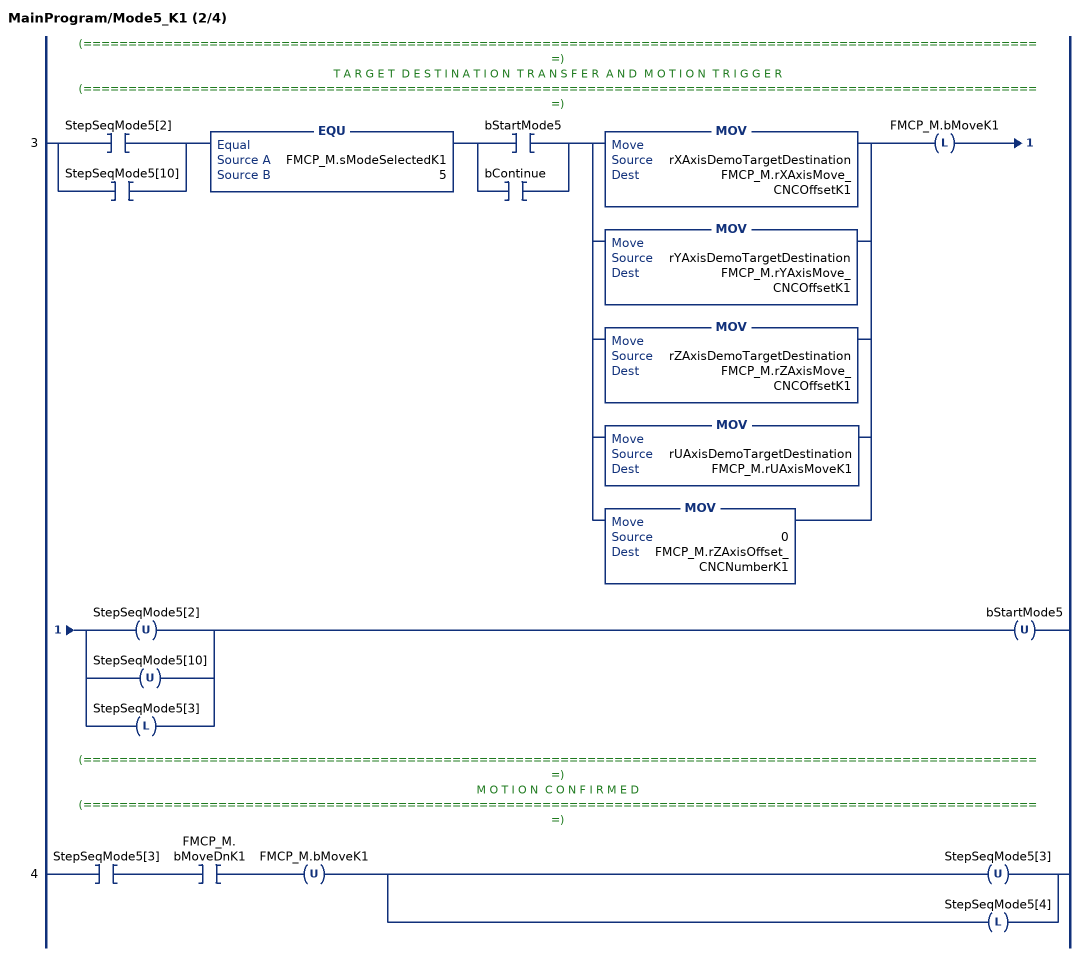
   // (===========================================================================================================)
   // T A R G E T  D E S T I N A T I O N  T R A N S F E R  A N D  M O T I O N  T R I G G E R
   // (===========================================================================================================)
   3: [XIC(StepSeqMode5[2]) ,XIC(StepSeqMode5[10]) ]EQU(FMCP_M.sModeSelectedK1,5)[XIC(bStartMode5) ,XIC(bContinue) ][MOV(rXAxisDemoTargetDestination,FMCP_M.rXAxisMove_CNCOffsetK1) ,MOV(rYAxisDemoTargetDestination,FMCP_M.rYAxisMove_CNCOffsetK1) ,MOV(rZAxisDemoTargetDestination,FMCP_M.rZAxisMove_CNCOffsetK1) ,MOV(rUAxisDemoTargetDestination,FMCP_M.rUAxisMoveK1) ,MOV(0,FMCP_M.rZAxisOffset_CNCNumberK1) ]OTL(FMCP_M.bMoveK1)[OTU(StepSeqMode5[2]) ,OTU(StepSeqMode5[10]) ,OTL(StepSeqMode5[3]) ]OTU(bStartMode5);
   // (===========================================================================================================)
   // M O T I O N  C O N F I R M E D
   // (===========================================================================================================)
   4: XIC(StepSeqMode5[3])XIC(FMCP_M.bMoveDnK1)OTU(FMCP_M.bMoveK1)[OTU(StepSeqMode5[3]) ,OTL(StepSeqMode5[4]) ];
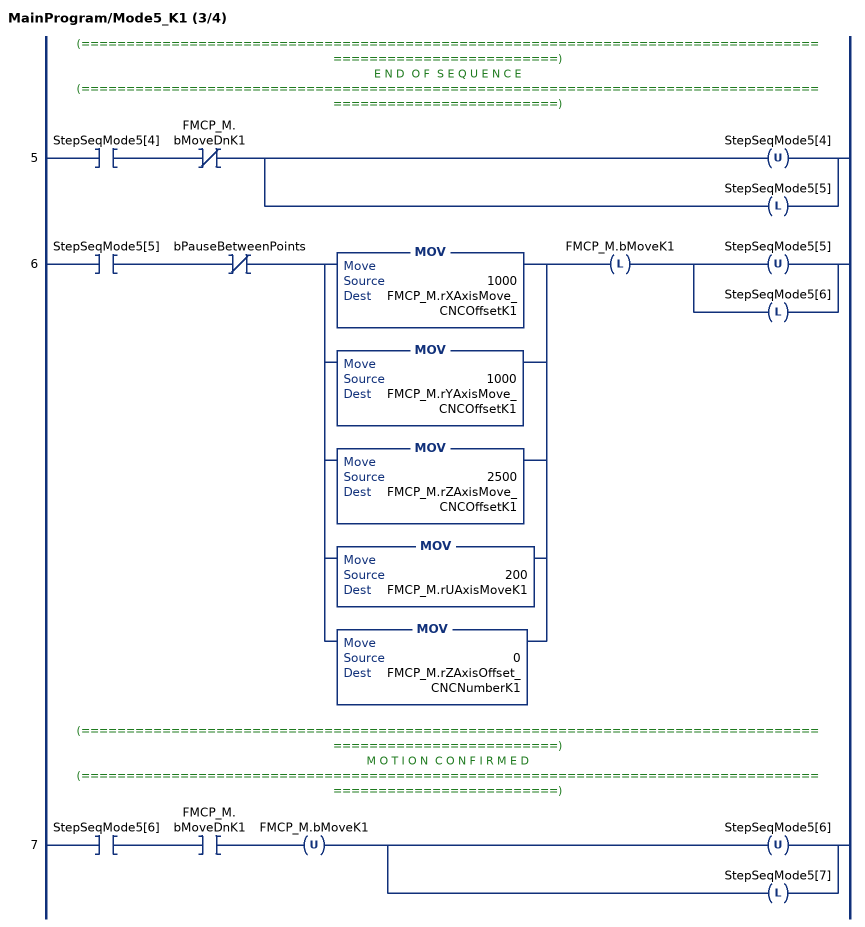
   // (===========================================================================================================)
   // E N D  O F  S E Q U E N C E
   // (===========================================================================================================)
   5: XIC(StepSeqMode5[4])XIO(FMCP_M.bMoveDnK1)[OTU(StepSeqMode5[4]) ,OTL(StepSeqMode5[5]) ];
   6: XIC(StepSeqMode5[5])XIO(bPauseBetweenPoints)[MOV(1000,FMCP_M.rXAxisMove_CNCOffsetK1) ,MOV(1000,FMCP_M.rYAxisMove_CNCOffsetK1) ,MOV(2500,FMCP_M.rZAxisMove_CNCOffsetK1) ,MOV(200,FMCP_M.rUAxisMoveK1) ,MOV(0,FMCP_M.rZAxisOffset_CNCNumberK1) ]OTL(FMCP_M.bMoveK1)[OTU(StepSeqMode5[5]) ,OTL(StepSeqMode5[6]) ];
   // (===========================================================================================================)
   // M O T I O N  C O N F I R M E D
   // (===========================================================================================================)
   7: XIC(StepSeqMode5[6])XIC(FMCP_M.bMoveDnK1)OTU(FMCP_M.bMoveK1)[OTU(StepSeqMode5[6]) ,OTL(StepSeqMode5[7]) ];
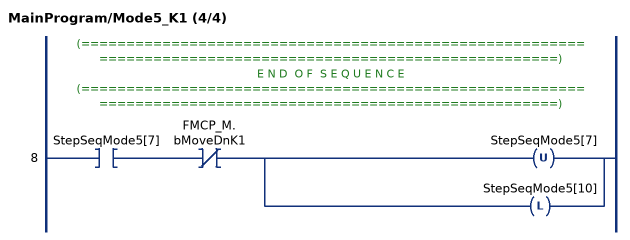
   // (===========================================================================================================)
   // E N D  O F  S E Q U E N C E
   // (===========================================================================================================)
   8: XIC(StepSeqMode5[7])XIO(FMCP_M.bMoveDnK1)[OTU(StepSeqMode5[7]) ,OTL(StepSeqMode5[10]) ];
END_ROUTINE

ROUTINE Mode6wOffset_K1   (* ladder *)
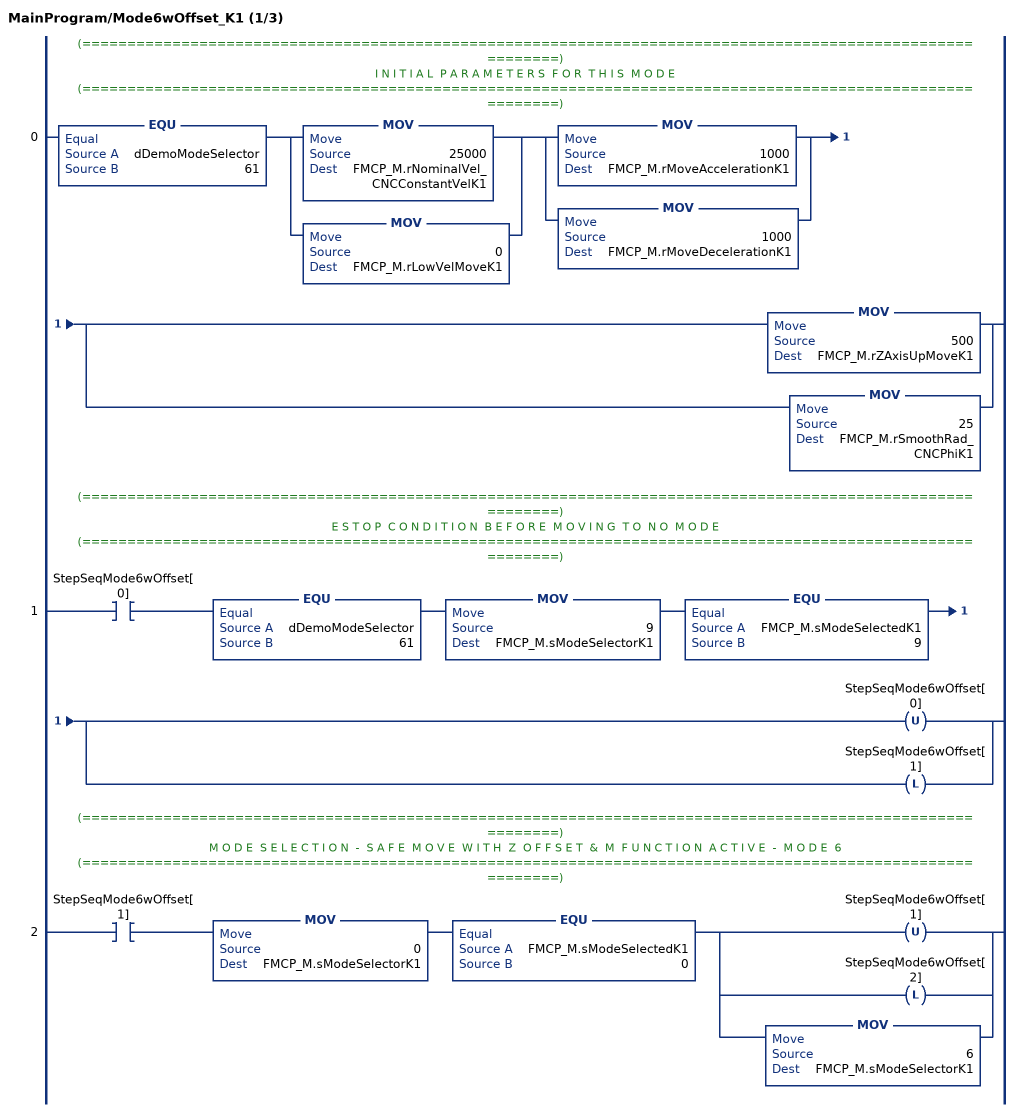
   // (===========================================================================================================)
   // I N I T I A L  P A R A M E T E R S  F O R  T H I S  M O D E
   // (===========================================================================================================)
   0: EQU(dDemoModeSelector,61)[MOV(25000,FMCP_M.rNominalVel_CNCConstantVelK1) ,MOV(0,FMCP_M.rLowVelMoveK1) ][MOV(1000,FMCP_M.rMoveAccelerationK1) ,MOV(1000,FMCP_M.rMoveDecelerationK1) ][MOV(500,FMCP_M.rZAxisUpMoveK1) ,MOV(25,FMCP_M.rSmoothRad_CNCPhiK1) ];
   // (===========================================================================================================)
   // E S T O P  C O N D I T I O N  B E F O R E  M O V I N G  T O  N O  M O D E
   // (===========================================================================================================)
   1: XIC(StepSeqMode6wOffset[0])EQU(dDemoModeSelector,61)MOV(9,FMCP_M.sModeSelectorK1)EQU(FMCP_M.sModeSelectedK1,9)[OTU(StepSeqMode6wOffset[0]) ,OTL(StepSeqMode6wOffset[1]) ];
   // (===========================================================================================================)
   // M O D E  S E L E C T I O N  -  S A F E  M O V E  W I T H  Z  O F F S E T  &  M  F U N C T I O N  A C T I V E  -  M O D E  6
   // (===========================================================================================================)
   2: XIC(StepSeqMode6wOffset[1])MOV(0,FMCP_M.sModeSelectorK1)EQU(FMCP_M.sModeSelectedK1,0)[OTU(StepSeqMode6wOffset[1]) ,OTL(StepSeqMode6wOffset[2]) ,MOV(6,FMCP_M.sModeSelectorK1) ];
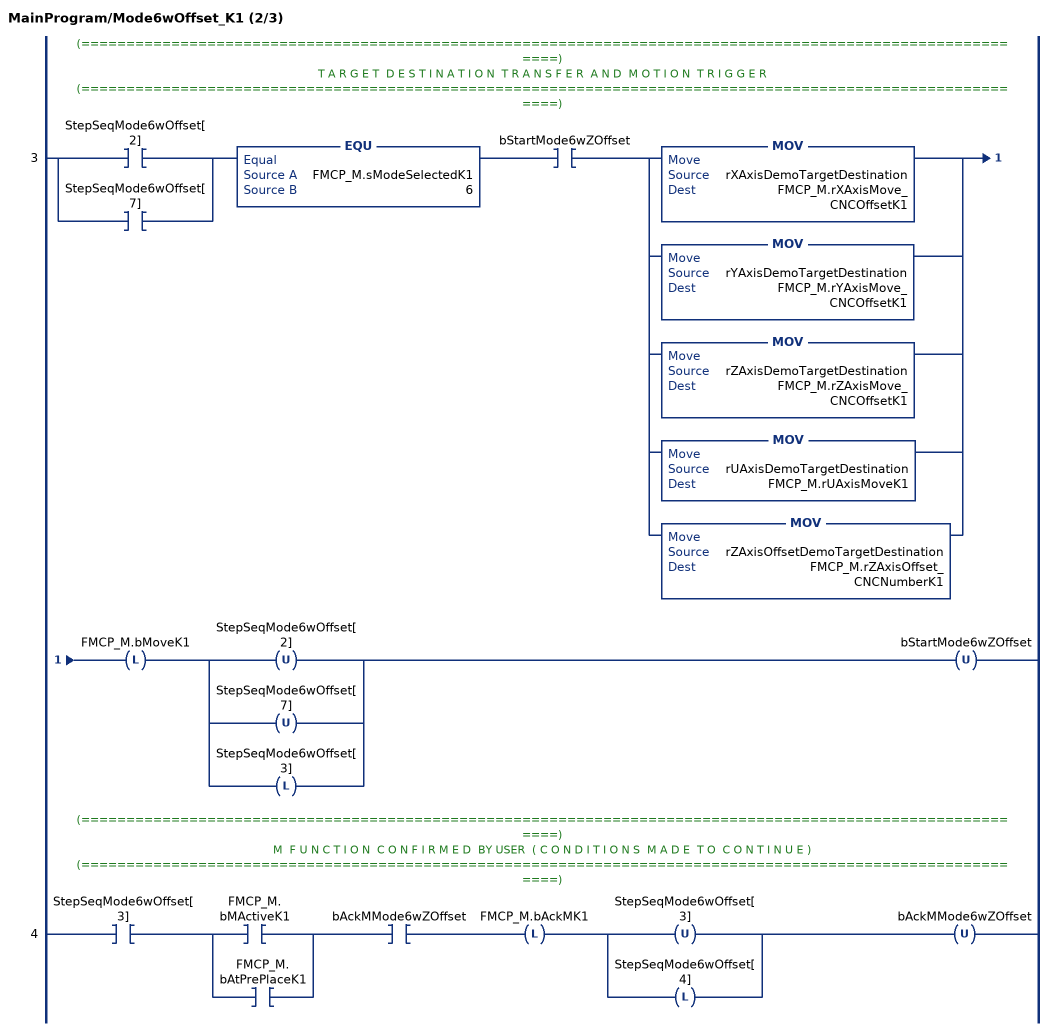
   // (===========================================================================================================)
   // T A R G E T  D E S T I N A T I O N  T R A N S F E R  A N D  M O T I O N  T R I G G E R
   // (===========================================================================================================)
   3: [XIC(StepSeqMode6wOffset[2]) ,XIC(StepSeqMode6wOffset[7]) ]EQU(FMCP_M.sModeSelectedK1,6)XIC(bStartMode6wZOffset)[MOV(rXAxisDemoTargetDestination,FMCP_M.rXAxisMove_CNCOffsetK1) ,MOV(rYAxisDemoTargetDestination,FMCP_M.rYAxisMove_CNCOffsetK1) ,MOV(rZAxisDemoTargetDestination,FMCP_M.rZAxisMove_CNCOffsetK1) ,MOV(rUAxisDemoTargetDestination,FMCP_M.rUAxisMoveK1) ,MOV(rZAxisOffsetDemoTargetDestination,FMCP_M.rZAxisOffset_CNCNumberK1) ]OTL(FMCP_M.bMoveK1)[OTU(StepSeqMode6wOffset[2]) ,OTU(StepSeqMode6wOffset[7]) ,OTL(StepSeqMode6wOffset[3]) ]OTU(bStartMode6wZOffset);
   // (===========================================================================================================)
   // M  F U N C T I O N  C O N F I R M E D  BY USER  ( C O N D I T I O N S  M A D E  T O  C O N T I N U E )
   // (===========================================================================================================)
   4: XIC(StepSeqMode6wOffset[3])[XIC(FMCP_M.bMActiveK1) ,XIC(FMCP_M.bAtPrePlaceK1) ]XIC(bAckMMode6wZOffset)OTL(FMCP_M.bAckMK1)[OTU(StepSeqMode6wOffset[3]) ,OTL(StepSeqMode6wOffset[4]) ]OTU(bAckMMode6wZOffset);
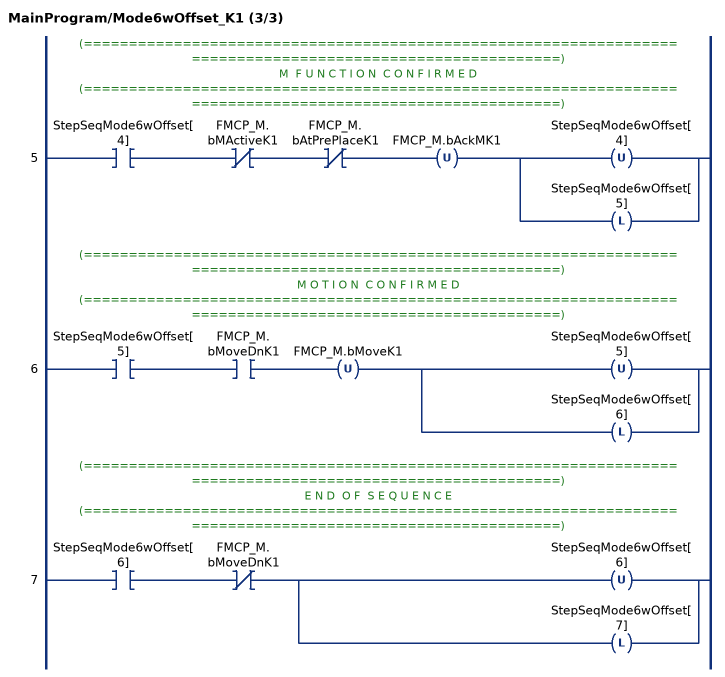
   // (===========================================================================================================)
   // M  F U N C T I O N  C O N F I R M E D
   // (===========================================================================================================)
   5: XIC(StepSeqMode6wOffset[4])XIO(FMCP_M.bMActiveK1)XIO(FMCP_M.bAtPrePlaceK1)OTU(FMCP_M.bAckMK1)[OTU(StepSeqMode6wOffset[4]) ,OTL(StepSeqMode6wOffset[5]) ];
   // (===========================================================================================================)
   // M O T I O N  C O N F I R M E D
   // (===========================================================================================================)
   6: XIC(StepSeqMode6wOffset[5])XIC(FMCP_M.bMoveDnK1)OTU(FMCP_M.bMoveK1)[OTU(StepSeqMode6wOffset[5]) ,OTL(StepSeqMode6wOffset[6]) ];
   // (===========================================================================================================)
   // E N D  O F  S E Q U E N C E
   // (===========================================================================================================)
   7: XIC(StepSeqMode6wOffset[6])XIO(FMCP_M.bMoveDnK1)[OTU(StepSeqMode6wOffset[6]) ,OTL(StepSeqMode6wOffset[7]) ];
END_ROUTINE

ROUTINE Mode6woOffset_K1   (* ladder *)
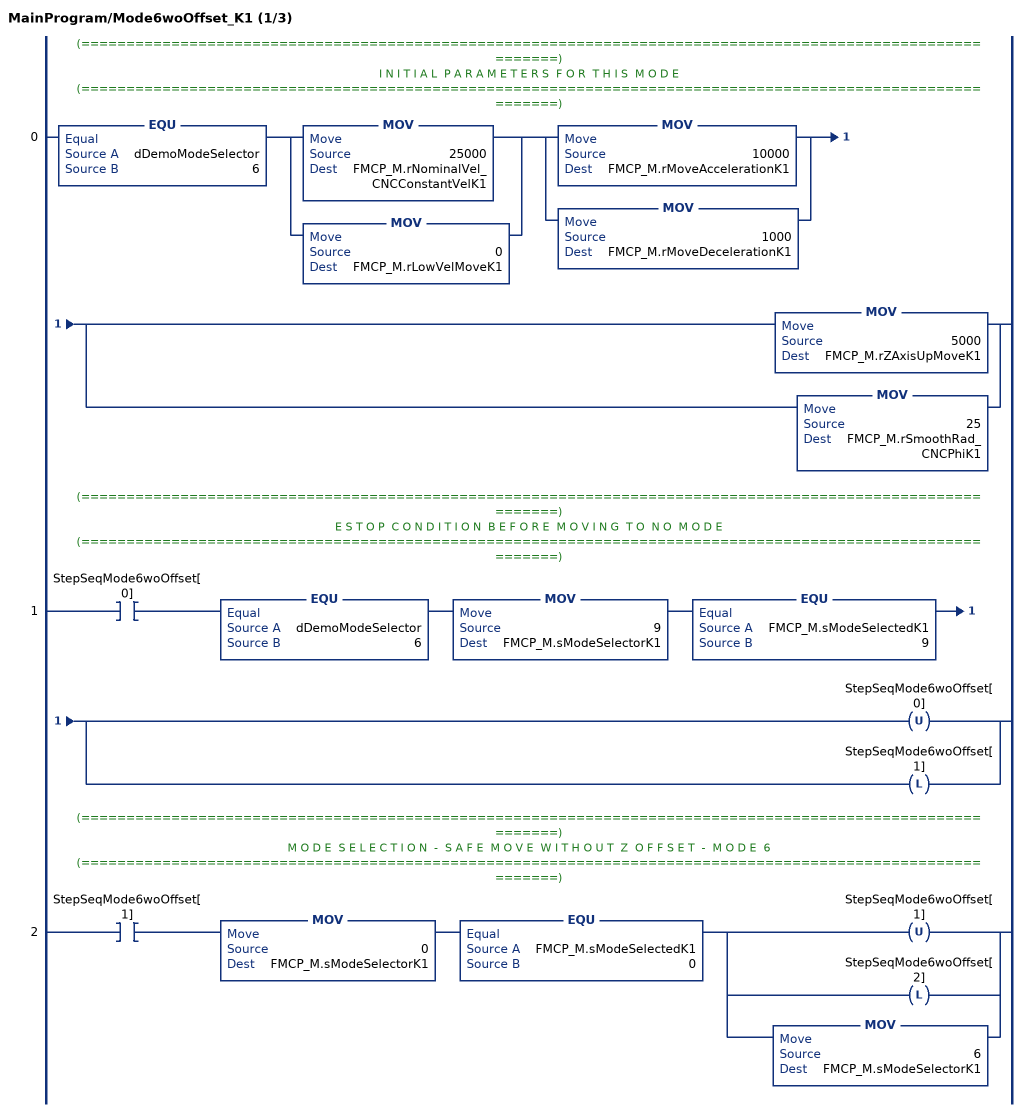
   // (===========================================================================================================)
   // I N I T I A L  P A R A M E T E R S  F O R  T H I S  M O D E
   // (===========================================================================================================)
   0: EQU(dDemoModeSelector,6)[MOV(25000,FMCP_M.rNominalVel_CNCConstantVelK1) ,MOV(0,FMCP_M.rLowVelMoveK1) ][MOV(10000,FMCP_M.rMoveAccelerationK1) ,MOV(1000,FMCP_M.rMoveDecelerationK1) ][MOV(5000,FMCP_M.rZAxisUpMoveK1) ,MOV(25,FMCP_M.rSmoothRad_CNCPhiK1) ];
   // (===========================================================================================================)
   // E S T O P  C O N D I T I O N  B E F O R E  M O V I N G  T O  N O  M O D E
   // (===========================================================================================================)
   1: XIC(StepSeqMode6woOffset[0])EQU(dDemoModeSelector,6)MOV(9,FMCP_M.sModeSelectorK1)EQU(FMCP_M.sModeSelectedK1,9)[OTU(StepSeqMode6woOffset[0]) ,OTL(StepSeqMode6woOffset[1]) ];
   // (===========================================================================================================)
   // M O D E  S E L E C T I O N  -  S A F E  M O V E  W I T H O U T  Z  O F F S E T  -  M O D E  6
   // (===========================================================================================================)
   2: XIC(StepSeqMode6woOffset[1])MOV(0,FMCP_M.sModeSelectorK1)EQU(FMCP_M.sModeSelectedK1,0)[OTU(StepSeqMode6woOffset[1]) ,OTL(StepSeqMode6woOffset[2]) ,MOV(6,FMCP_M.sModeSelectorK1) ];
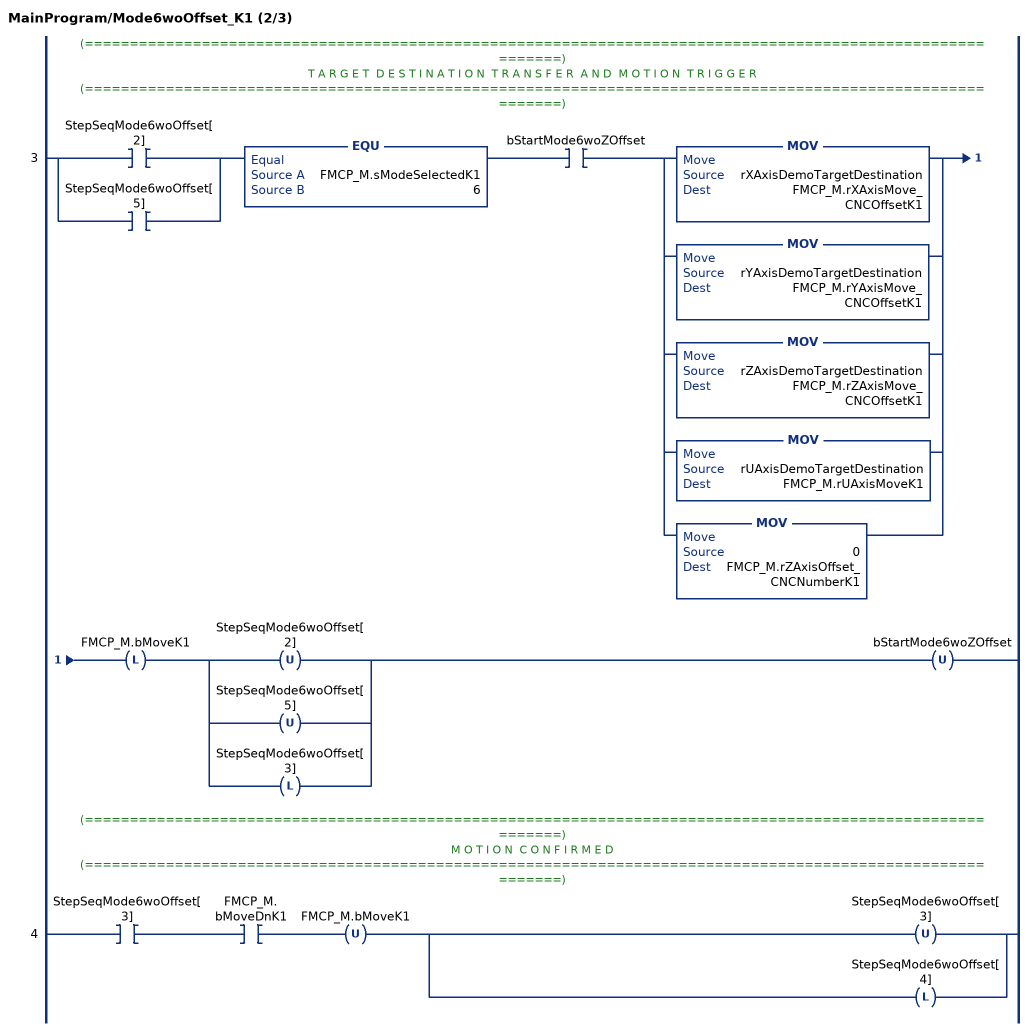
   // (===========================================================================================================)
   // T A R G E T  D E S T I N A T I O N  T R A N S F E R  A N D  M O T I O N  T R I G G E R
   // (===========================================================================================================)
   3: [XIC(StepSeqMode6woOffset[2]) ,XIC(StepSeqMode6woOffset[5]) ]EQU(FMCP_M.sModeSelectedK1,6)XIC(bStartMode6woZOffset)[MOV(rXAxisDemoTargetDestination,FMCP_M.rXAxisMove_CNCOffsetK1) ,MOV(rYAxisDemoTargetDestination,FMCP_M.rYAxisMove_CNCOffsetK1) ,MOV(rZAxisDemoTargetDestination,FMCP_M.rZAxisMove_CNCOffsetK1) ,MOV(rUAxisDemoTargetDestination,FMCP_M.rUAxisMoveK1) ,MOV(0,FMCP_M.rZAxisOffset_CNCNumberK1) ]OTL(FMCP_M.bMoveK1)[OTU(StepSeqMode6woOffset[2]) ,OTU(StepSeqMode6woOffset[5]) ,OTL(StepSeqMode6woOffset[3]) ]OTU(bStartMode6woZOffset);
   // (===========================================================================================================)
   // M O T I O N  C O N F I R M E D
   // (===========================================================================================================)
   4: XIC(StepSeqMode6woOffset[3])XIC(FMCP_M.bMoveDnK1)OTU(FMCP_M.bMoveK1)[OTU(StepSeqMode6woOffset[3]) ,OTL(StepSeqMode6woOffset[4]) ];
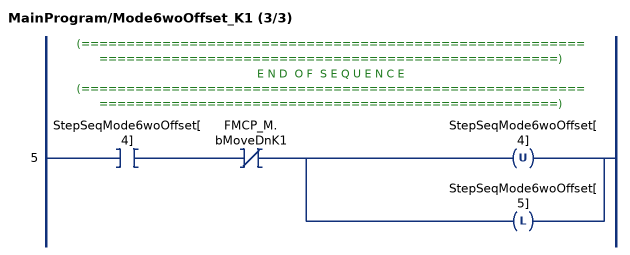
   // (===========================================================================================================)
   // E N D  O F  S E Q U E N C E
   // (===========================================================================================================)
   5: XIC(StepSeqMode6woOffset[4])XIO(FMCP_M.bMoveDnK1)[OTU(StepSeqMode6woOffset[4]) ,OTL(StepSeqMode6woOffset[5]) ];
END_ROUTINE

ROUTINE Mode7CNC_K1   (* ladder *)
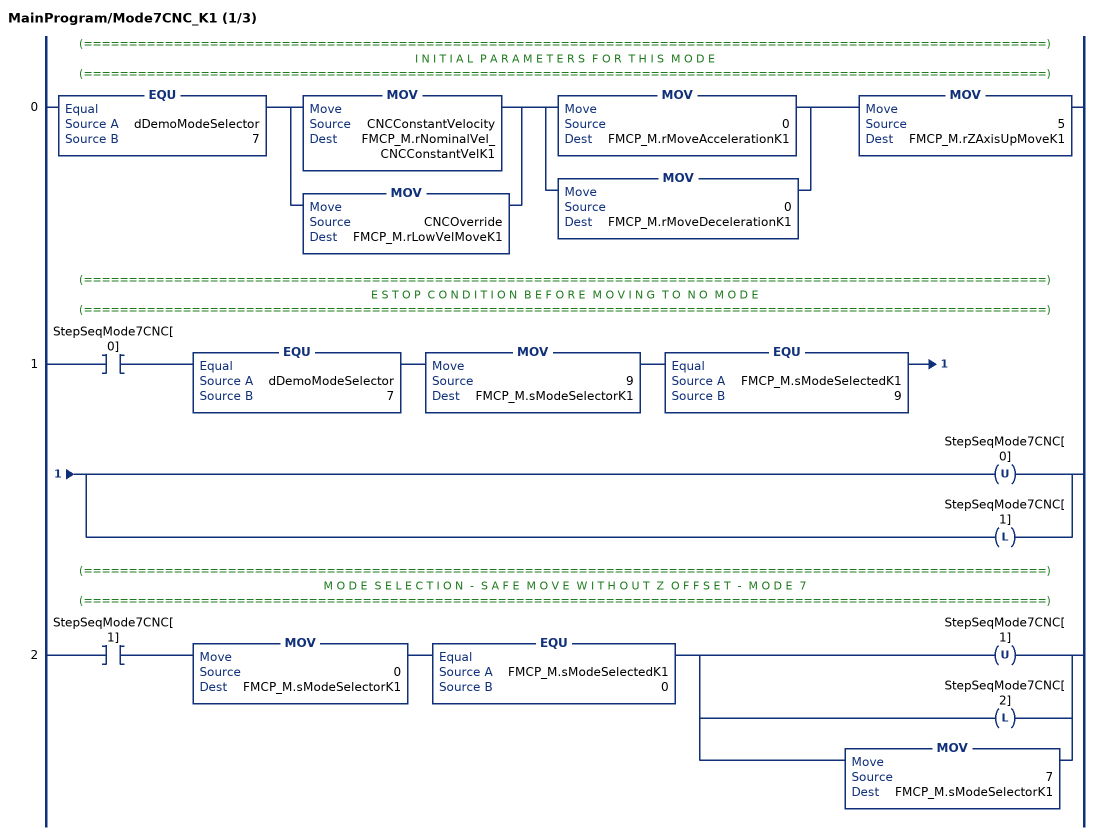
   // (===========================================================================================================)
   // I N I T I A L  P A R A M E T E R S  F O R  T H I S  M O D E
   // (===========================================================================================================)
   0: EQU(dDemoModeSelector,7)[MOV(CNCConstantVelocity,FMCP_M.rNominalVel_CNCConstantVelK1) ,MOV(CNCOverride,FMCP_M.rLowVelMoveK1) ][MOV(0,FMCP_M.rMoveAccelerationK1) ,MOV(0,FMCP_M.rMoveDecelerationK1) ]MOV(5,FMCP_M.rZAxisUpMoveK1);
   // (===========================================================================================================)
   // E S T O P  C O N D I T I O N  B E F O R E  M O V I N G  T O  N O  M O D E
   // (===========================================================================================================)
   1: XIC(StepSeqMode7CNC[0])EQU(dDemoModeSelector,7)MOV(9,FMCP_M.sModeSelectorK1)EQU(FMCP_M.sModeSelectedK1,9)[OTU(StepSeqMode7CNC[0]) ,OTL(StepSeqMode7CNC[1]) ];
   // (===========================================================================================================)
   // M O D E  S E L E C T I O N  -  S A F E  M O V E  W I T H O U T  Z  O F F S E T  -  M O D E  7
   // (===========================================================================================================)
   2: XIC(StepSeqMode7CNC[1])MOV(0,FMCP_M.sModeSelectorK1)EQU(FMCP_M.sModeSelectedK1,0)[OTU(StepSeqMode7CNC[1]) ,OTL(StepSeqMode7CNC[2]) ,MOV(7,FMCP_M.sModeSelectorK1) ];
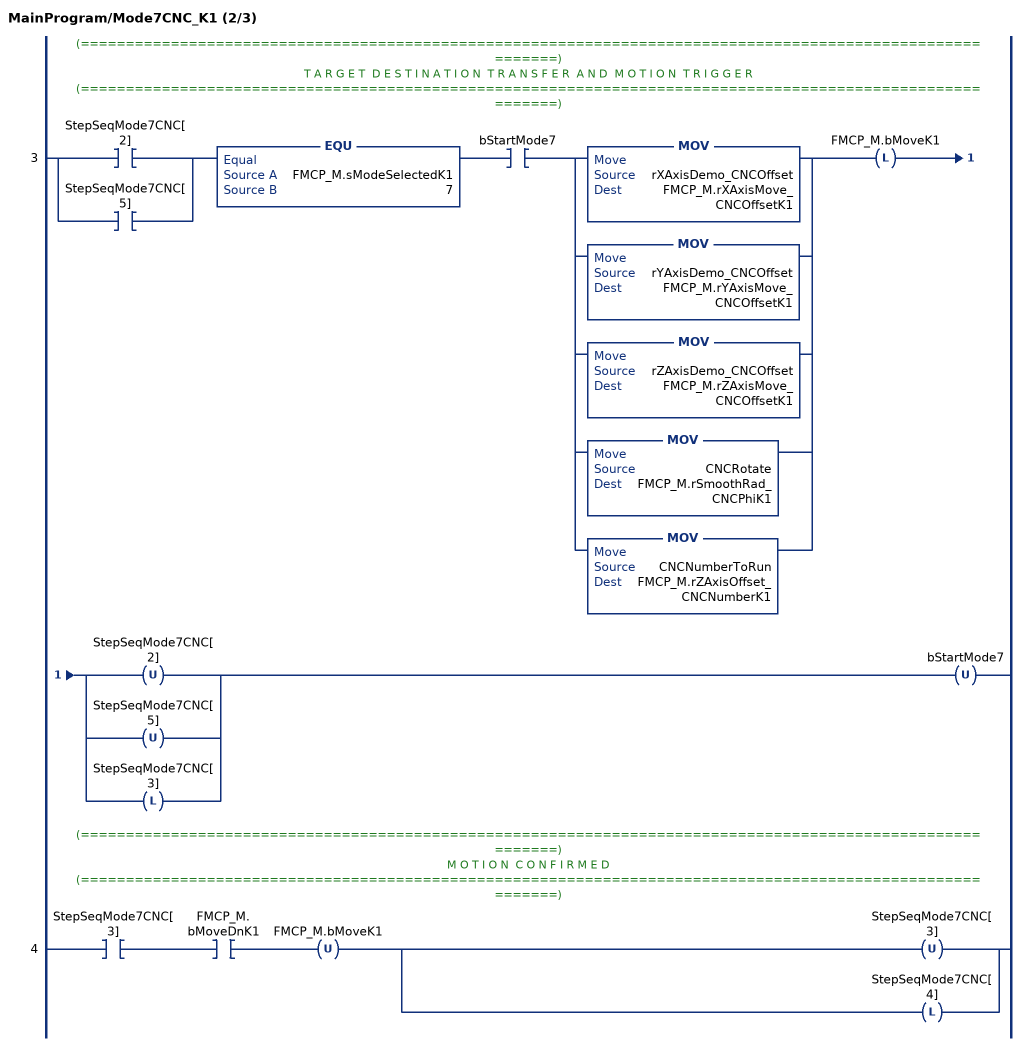
   // (===========================================================================================================)
   // T A R G E T  D E S T I N A T I O N  T R A N S F E R  A N D  M O T I O N  T R I G G E R
   // (===========================================================================================================)
   3: [XIC(StepSeqMode7CNC[2]) ,XIC(StepSeqMode7CNC[5]) ]EQU(FMCP_M.sModeSelectedK1,7)XIC(bStartMode7)[MOV(rXAxisDemo_CNCOffset,FMCP_M.rXAxisMove_CNCOffsetK1) ,MOV(rYAxisDemo_CNCOffset,FMCP_M.rYAxisMove_CNCOffsetK1) ,MOV(rZAxisDemo_CNCOffset,FMCP_M.rZAxisMove_CNCOffsetK1) ,MOV(CNCRotate,FMCP_M.rSmoothRad_CNCPhiK1) ,MOV(CNCNumberToRun,FMCP_M.rZAxisOffset_CNCNumberK1) ]OTL(FMCP_M.bMoveK1)[OTU(StepSeqMode7CNC[2]) ,OTU(StepSeqMode7CNC[5]) ,OTL(StepSeqMode7CNC[3]) ]OTU(bStartMode7);
   // (===========================================================================================================)
   // M O T I O N  C O N F I R M E D
   // (===========================================================================================================)
   4: XIC(StepSeqMode7CNC[3])XIC(FMCP_M.bMoveDnK1)OTU(FMCP_M.bMoveK1)[OTU(StepSeqMode7CNC[3]) ,OTL(StepSeqMode7CNC[4]) ];
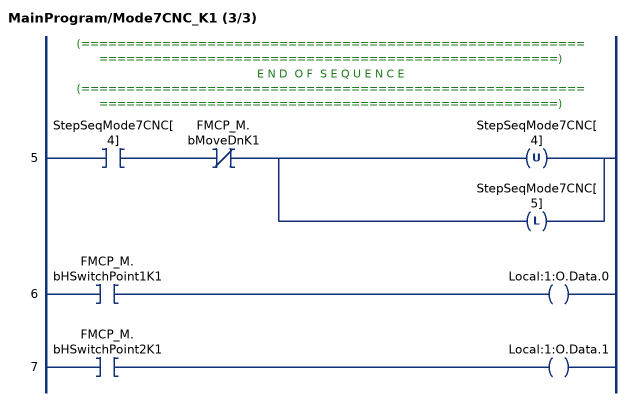
   // (===========================================================================================================)
   // E N D  O F  S E Q U E N C E
   // (===========================================================================================================)
   5: XIC(StepSeqMode7CNC[4])XIO(FMCP_M.bMoveDnK1)[OTU(StepSeqMode7CNC[4]) ,OTL(StepSeqMode7CNC[5]) ];
   6: XIC(FMCP_M.bHSwitchPoint1K1)OTE(Local:1:O.Data.0);
   7: XIC(FMCP_M.bHSwitchPoint2K1)OTE(Local:1:O.Data.1);
END_ROUTINE
END_PROGRAM
